// TIA Portal V15.1 export
// export: Created 2024-06-21T08:41:02.6727336Z, ExportSetting WithDefaults, DisplayName Totally Integrated Automation Portal, DisplayVersion V15.1 Update 5, DisplayName TIA Portal Openness, DisplayVersion V15.1 Update 5, DisplayName SINAMICS Startdrive Advanced, DisplayVersion V15.1, DisplayName G130, G150, S120, S150, SINAMICS MV, S210, DisplayVersion V15.1, DisplayName G110M, G120, G120C, G120D, G120P, DisplayVersion V15.1, DisplayName STEP 7 Professional, DisplayVersion V15.1 Update 5, DisplayName STEP 7 Safety, DisplayVersion V15.1, DisplayName WinCC Professional, DisplayVersion V15.1 Update 5, DisplayName SIMATIC Visualization Architect, DisplayVersion V15.1
FUNCTION_BLOCK "LProcDiffAI"   // FB1705, FBD
TITLE = LProcDiffAI
{ S7_Optimized_Access := 'FALSE' }
AUTHOR : VCC
FAMILY : Control
NAME : DiffAI
VERSION : 0.1
// ================================================================================
// DiffAI is used when a comparasion between two analog input signals is wanted to
// verify that the signals differ from each other more than the accepted 
// difference.
// ================================================================================
// stored: AutoNumber false, IsIECCheckEnabled false, SetENOAutomatically False, UDAEnableTagReadback false
   VAR_INPUT
      I_AnalogIn1 { ExternalAccessible := 'False'; ExternalVisible := 'False'; ExternalWritable := 'False'} : Real;   // Analog signal 1 to compare
      I_AnalogIn2 { ExternalAccessible := 'False'; ExternalVisible := 'False'; ExternalWritable := 'False'} : Real;   // Analog signal 2 to compare
      I_MaxDifference { ExternalAccessible := 'False'; ExternalVisible := 'False'; ExternalWritable := 'False'} : Real;   // Maximal accepted difference in %
   END_VAR
   VAR_OUTPUT
      O_DifferAI { ExternalAccessible := 'False'; ExternalVisible := 'False'; ExternalWritable := 'False'} : Bool;   // The two analog signals differ
   END_VAR
   VAR DB_SPECIFIC
      MaxDiffPercent { ExternalAccessible := 'False'; ExternalVisible := 'False'; ExternalWritable := 'False'} : Real;   // Maximal accepted difference in %
      Subtract { ExternalAccessible := 'False'; ExternalVisible := 'False'; ExternalWritable := 'False'} : Real;   // Analog inputs subtracted
      SubtractABS { ExternalAccessible := 'False'; ExternalVisible := 'False'; ExternalWritable := 'False'} : Real;   // ABS-value for subtracted Analog inputs
      DiffCalc { ExternalAccessible := 'False'; ExternalVisible := 'False'; ExternalWritable := 'False'} : Real;   // Calculated Difference
      DiffPercent { ExternalAccessible := 'False'; ExternalVisible := 'False'; ExternalWritable := 'False'} : Real;   // Difference between inputs %
   END_VAR
BEGIN

REGION Network 1: **** 1 - Inputs **** Maximal accepted difference in %
   // Maximal accepted difference in %
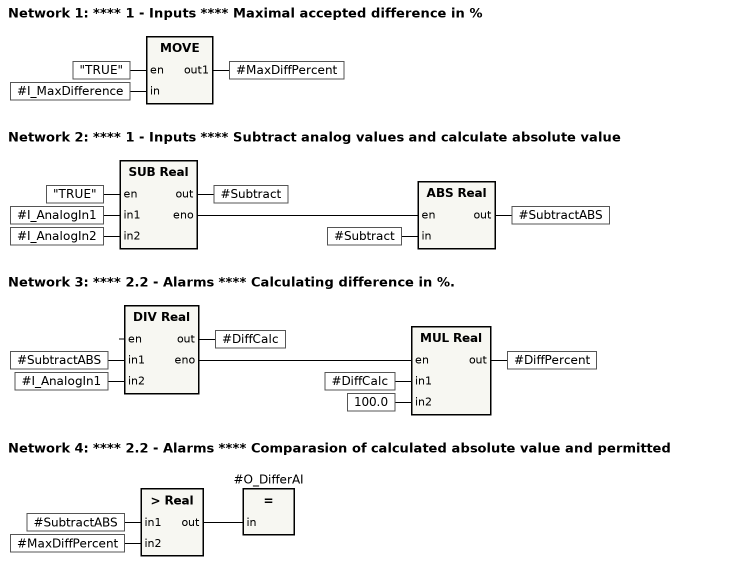
   IF "TRUE" THEN #MaxDiffPercent := #I_MaxDifference; END_IF;
END_REGION

REGION Network 2: **** 1 - Inputs **** Subtract analog values and calculate absolute value
   // Subtract analog values and calculate absolute value
   // ENO of a box is taken as its EN; it also drops when the box reports an error
   IF "TRUE" THEN
       #Subtract := #I_AnalogIn1 - #I_AnalogIn2;
       #SubtractABS := ABS(#Subtract);
   END_IF;
END_REGION

REGION Network 3: **** 2.2 - Alarms **** Calculating difference in %.
   // Calculating difference in %.
   // ENO of a box is taken as its EN; it also drops when the box reports an error
   #DiffCalc := #SubtractABS / #I_AnalogIn1;
   #DiffPercent := #DiffCalc * 100.0;
END_REGION

REGION Network 4: **** 2.2 - Alarms **** Comparasion of calculated absolute value and permitted
   // Alarm generation: Comparasion of calculated absolute value and permitted 
   // difference
   #O_DifferAI := #SubtractABS > #MaxDiffPercent;
END_REGION
END_FUNCTION_BLOCK
